// TwinCAT 3 PLC project Simulator
// ProgramVersion: 3.1.4023.0
// libraries:
//   Tc2_Standard, * (Beckhoff Automation GmbH)
//   Tc2_System, * (Beckhoff Automation GmbH)
//   Tc3_Module, * (Beckhoff Automation GmbH)
// project tree:
//   / PlcTask.TcTTO
//   01_Application/ MAIN.TcPOU
// (motion and I/O tree: see PLC project machinea)
// real-time tasks:
//   TASK PlcTask: cycle T#10ms, priority 20, ADS port 350
//   TASK PlcTask1: cycle T#10ms, priority 21, ADS port 351
// variable links:
//   MachineA/MachineA Instance <-> Simulator/Simulator Instance
//     PlcTask Inputs/MAIN.fbMachine.fbArm.fbFrontSensor.bDetect <-> PlcTask Outputs/MAIN.bFrontSensor
//     PlcTask Inputs/MAIN.fbMachine.fbArm.fbHomeSensor.bDetect <-> PlcTask Outputs/MAIN.bHomeSensor
//     PlcTask Inputs/MAIN.fbMachine.fbArm.fbRearSensor.bDetect <-> PlcTask Outputs/MAIN.bRearSensor
//     PlcTask Outputs/MAIN.fbMachine.fbArm.fbInverter.bClockwise <-> PlcTask Inputs/MAIN.bClockwise
//     PlcTask Outputs/MAIN.fbMachine.fbArm.fbInverter.bCounterClockwise <-> PlcTask Inputs/MAIN.bCounterClockwise
//     PlcTask Outputs/MAIN.fbMachine.fbArm.fbInverter.rAnalogSV <-> PlcTask Inputs/MAIN.rAnalogSV

CONFIGURATION Simulator
    RESOURCE PLC ON TwinCAT3
        TASK PlcTask(INTERVAL := T#10ms, PRIORITY := 21);
        PROGRAM MAIN WITH PlcTask : MAIN;
    END_RESOURCE
END_CONFIGURATION

// ---- 01_Application/MAIN.TcPOU
PROGRAM MAIN
VAR
	bFrontSensor			AT %Q* : BOOL;
	bHomeSensor				AT %Q* : BOOL;
	bRearSensor				AT %Q* : BOOL;
	
	//rAnalogPV				AT %Q* : REAL;
	rAnalogSV				AT %I* : REAL;
	
	rAxisPV					AT %Q* : REAL;
	//rAxisSV					AT %I* : REAL;
	
	bClockwise				AT %I* : BOOL;
	bCounterClockwise		AT %I* : BOOL;
	
	//rAccelerationSV			AT %I* : REAL;
	//rDecelerationSV			AT %I* : REAL;
END_VAR

IF rAxisPV > -10 AND rAxisPV < -9 THEN
	bFrontSensor := TRUE;
ELSE
	bFrontSensor := FALSE;
END_IF

IF rAxisPV > 9 AND rAxisPV < 10 THEN
	bHomeSensor := TRUE;
ELSE
	bHomeSensor := FALSE;
END_IF

IF rAxisPV > 59 AND rAxisPV < 60 THEN
	bRearSensor := TRUE;
ELSE
	bRearSensor := FALSE;
END_IF


IF bClockwise THEN
	rAxisPV := rAxisPV - rAnalogSV;
ELSIF bCounterClockwise THEN
	rAxisPV := rAxisPV + rAnalogSV;
END_IF

END_PROGRAM
